Staubli VAL3: cmdEnableHold.pgx

public program cmdEnableHold(num x_nAxNum (dimensions=1))
begin
  // this program issues an 'Enable Hold'  command to the selected drive.
  // This bit must be set to enable drive power
  //发送“enable hold”指令到所选控制器
  //用于设置驱动器电源开启
  //  doEnableHold[x_nAxNum]=true
end
